FUNCTION_BLOCK E_FB_DELAY (* Delayed event propagation *)
  (* Standard: 61499-1 Annex A; Description: Copyright (c) 2017 fortiss GmbH This program and the accompanying materials are made available under the terms of the Eclipse Public License 2.0 which is available at https://www.eclipse.org/legal/epl-2.0/ SPDX-License-Identifier: EPL-2.0 *)
  (* Version 3.1, 2026-08-14, Franz Höpfinger, HR Agrartechnik GmbH, FB_TON like cyclic Interface *)
  (* Version 3.0, 2025-04-14, Patrick Aigner, changed package *)
  (* Version 1.0, 2017-09-21, Alois Zoitl, fortiss GmbH, initial API and implementation and/or initial documentation *)
  PACKAGE adapter::events::TimeOut;
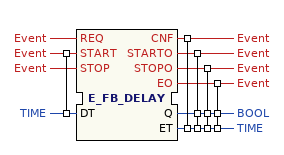
  EVENT_INPUT
    REQ; (* Normal Execution Request *)
    START WITH DT; (* Start delayed event propagation *)
    STOP; (* Stop the delayed event propagation *)
  END_EVENT
  EVENT_OUTPUT
    CNF WITH ET; (* Execution Confirmation *)
    STARTO WITH Q, ET;
    STOPO WITH Q, ET;
    EO WITH Q, ET; (* Delayed event *)
  END_EVENT
  VAR_INPUT
    DT : TIME; (* Delay time, >0 *)
  END_VAR
  VAR_OUTPUT
    Q : BOOL; (* Output is started = TRUE *)
    ET : TIME; (* Elapsed time *)
  END_VAR
  VAR
    StartTime : TIME;
  END_VAR
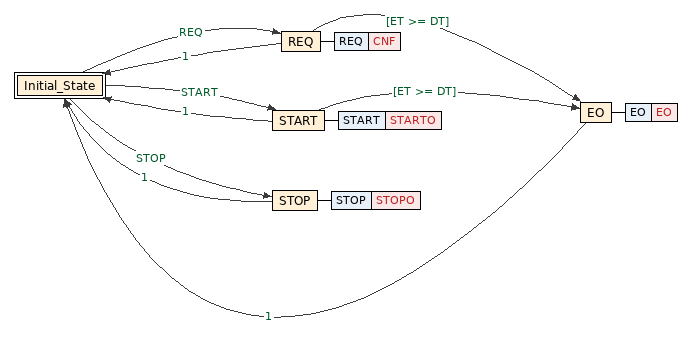
  EC_STATES
    Initial_State; (* Initial State *)
    REQ : REQ -> CNF;
    START : START -> STARTO;
    STOP : STOP -> STOPO;
    EO : EO -> EO;
  END_STATES
  EC_TRANSITIONS
    Initial_State TO REQ := REQ;
    Initial_State TO START := START;
    Initial_State TO STOP := STOP;
    REQ TO EO := [ET >= DT];
    REQ TO Initial_State := 1;
    STOP TO Initial_State := 1;
    START TO EO := [ET >= DT];
    START TO Initial_State := 1;
    EO TO Initial_State := 1;
  END_TRANSITIONS
  ALGORITHM REQ IN ST: (* Poll elapsed time while armed (Q=TRUE); no-op otherwise. Meant to be driven cyclically (e.g. by an external E_CYCLE) so ET stays live while the delay is running. *)
VAR_TEMP
	SysTime : TIME;
END_VAR
IF Q THEN
	SysTime := NOW_MONOTONIC();
	ET := SysTime - StartTime;
END_IF;
  END_ALGORITHM
  ALGORITHM START IN ST: (* Arm the timer: record the start time, reset ET to 0 and set Q=TRUE so REQ begins advancing ET. *)
StartTime := NOW_MONOTONIC();
Q := BOOL#TRUE;
ET := T#0s;
  END_ALGORITHM
  ALGORITHM STOP IN ST: (* Cancel the timer without firing EO: clear Q and reset ET to 0. *)
Q := BOOL#FALSE;
ET := T#0s;
  END_ALGORITHM
  ALGORITHM EO IN ST: (* Runs once when ET reaches DT (via the REQ/START -> EO transition). Clears Q and resets ET to 0, so ET stays below DT until the next START - a later REQ can no longer re-satisfy [ET>=DT] and re-fire EO. *)
Q := BOOL#FALSE;
ET := T#0s;
  END_ALGORITHM
END_FUNCTION_BLOCK
